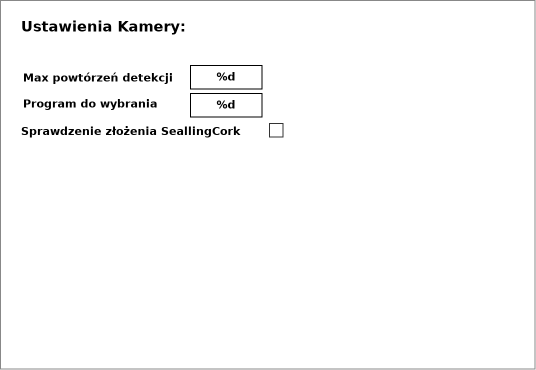
VISUALIZATION vSonicPress_SubVision  // 536x370
VAR_IN_OUT
	fbMachine: fbSonicPress;
END_VAR
    Label (20,66 169x24), "Max powtórzeń detekcji"
    Rectangle (190,65 72x24), "%d", text variable: MAIN.fbS01_KeyencePNVisSens.stParams.iMaxTrigRepeats, input disabled if: NOT GVL.fbUserLogin.bPermissionGranted
        OnMouseClick: write the text variable via Default, min 0, max 6
    Label (262,64 42x24)
    Label (262,91 42x24)
    Label (20,92 169x24), "Program do wybrania"
    Rectangle (190,93 72x24), "%d", text variable: MAIN.fbS01_KeyencePNVisSens.stParams.iProgramNumber, input disabled if: NOT GVL.fbUserLogin.bPermissionGranted
        OnMouseClick: write the text variable via Default, min 0, max 10, title 'Trigger position'
    Label (18,10 271x33), "Ustawienia Kamery:"
    Checkbox (267,117 26x26), variable: MAIN.fbS01_KeyencePNVisSens.stParams.bInspectionEnable, input disabled if: GVL.fbUserLogin.nUserRole <> nSQL_UserRoles.Maintenance
    Label (18,114 225x35), "Sprawdzenie złożenia SeallingCork"
END_VISUALIZATION

(* stored: Version 1.1.0.1, ProductVersion 3.1.4024.13
   Visu vSonicPress_SubVision: Id {17d84caf-6f2b-47bc-bd40-26319ec1b9e1} *)
